FUNCTION F_AlyTimestampToDCTimestruct : DCTIMESTRUCT
VAR_INPUT
	tTimestamp: ULINT;
END_VAR
VAR
	tFileTime: T_FILETIME;
	newDCTime: T_DCTIME64;
	
	fbToLocal: FB_FileTimeToTzSpecificLocalTime;
	//Malay Peninsula Daylight Time
	//(UTC+08:00) Kuala Lumpur, Singapore
	tzInfo: ST_TimeZoneInformation := (bias := -480);
END_VAR

tFileTime:= DCTIME64_TO_Filetime(tTimestamp);
fbToLocal(in:= tFileTime, tzInfo:= tzInfo);
newDCTime:= FILETIME_TO_DCTIME64(fbToLocal.out);

F_AlyTimestampToDCTimestruct:= DCTIME64_TO_DCTIMESTRUCT(newDCTime);

END_FUNCTION

(* stored: POU F_AlyTimestampToDCTimestruct: Id 6acace79-ea17-4c2c-80cc-8e98e2ae707e, SpecialFunc None *)
